
(* ===== HMI "HiddenHmiRTDeviceFaceplateTypes" =====

HMI tags "950e3fec-f6dc-4982-844c-a829a90ca654"
   "ExtProg" : 34deb92b-2d19-457e-81d5-55f2b3080f0d, internal
*)

(* ===== HMI "HiddenHmiRTDeviceFaceplateTypes" =====

HMI tags "9ca7d841-4e4d-4293-b7f5-7bf308eb5ab1"
   "ExtProg" : 34deb92b-2d19-457e-81d5-55f2b3080f0d, internal
*)

(* ===== HMI "HMI_RT_1" =====

HMI tags "WinProgManager"
   "_WINPROGMANAGER_" : 34deb92b-2d19-457e-81d5-55f2b3080f0d, internal
*)